FUNCTION_BLOCK ClampCPLinPPR EXTENDS ClearpathPositionLinPPR
VAR_INPUT
	PartPresentHi AT %I* : BOOL;
	PartPresentLo AT %I* : BOOL;
END_VAR
VAR_OUTPUT
	PartPresent_PO	: BOOL;
	PartPresent_VO	: BOOL;
	HomeStatusMsg_VO : string;	
END_VAR
VAR
	ClampHomeCase : INT;
END_VAR


IF Mode_PI =1 THEN //autohoming in automode
	CASE ClampHomeCase OF
		0:  
			IF Out.Homed_PO =0 AND PartPresentHi =0 AND PartPresentLo=0 THEN
			 ClampHomeCase :=20;
			END_IF
			IF Out.Homed_PO =0 AND PartPresentHi =1 AND PartPresentLo =1 THEN
			//Part in clamp set home at xx distance and set home
			ClampHomeCase:=10;
			END_IF
		10: //use psudeo home against part pipes
			Out.Homed_PO:=1;
			HomeCase:=0;
			Out.DistancePos_PO:=120;
			pulsecount :=120; //dis *2 (2 ppr per dis on base)
			expectedPulse :=120; //dis *2 (2 ppr per dis on base)
			Out.ExpDistancePos_PO :=120;
			ClampHomeCase:=0;
		20: //Use clamp home start
			bHomeStart_PI :=1;
			IF Out.Homed_PO THEN 
				ClampHomeCase:=0;
			END_IF
		
		30: //only one partpresnt is on.  Home, exetend and try again or flip error code
			ClampHomeCase:=0;
			HomeStatusMsg_VO:='homing not possible only one part present sensor is on. Manual reset req';
		
	END_CASE
	
END_IF

END_FUNCTION_BLOCK

(* stored: Version 1.1.0.1, ProductVersion 3.1.4024.11
   POU ClampCPLinPPR: Id {289dd517-9f11-427f-a240-c90e875ba3c1}, SpecialFunc None *)
